Omron CX-Programmer project NewProject (CX-Programmer 9.75)

# PLC NewPLC1: CJ2M CPU31
I/O table (CPU CJ2M-CPU31): rack 0 slot 11 CJ2M-EIP21

## Global symbols (name address type ; comment)
0.00 BOOL  ; SW1
0.01 BOOL  ; CAPACITIVE 2
0.02 BOOL  ; CAPACITIVE 3
0.04 BOOL  ; INDUCTIVE SENSOR
0.13 BOOL  ; REEST PASS DENY
0.14 BOOL  ; RESET ACCESSS
0.15 BOOL  ; RESET ACCESS
10.00 BOOL  ; SW1
10.01 BOOL  ; SW2
10.02 BOOL  ; SW3
10.03 BOOL  ; SW4
10.04 BOOL  ; RESET
10.05 BOOL  ; START
10.06 BOOL  ; STOP
1.00 BOOL  ; MAS
1.01 BOOL  ; LED
1.02 BOOL  ; ACUATOR
1.03 BOOL  ; INDUCTIVE OUTPUT
1.04 BOOL  ; GREEN LIGHT
1.05 BOOL  ; RED LIGHT
1.07 BOOL  ; NOT MAS
1.08 BOOL  ; KA sw
1.15 BOOL  ; ACCESS DENIED
20.00 BOOL  ; K1
20.01 BOOL  ; K3
20.02 BOOL  ; K2
20.03 BOOL  ; K4
20.04 BOOL  ; ACCESS GRANTED
20.05 BOOL  ; KEEP 1
20.06 BOOL  ; KEEP SW2
30.00 BOOL  ; KS1
30.01 BOOL  ; KS2
30.02 BOOL  ; KS3
30.03 BOOL  ; KS4
40.00 BOOL  ; KA
40.01 BOOL  ; KB
40.02 BOOL  ; KC
40.03 BOOL  ; KD
40.04 BOOL  ; KEEP LIGHT1
C0000 BOOL  ; COUNTER PEPLE
C1 CHANNEL  ; compare

## Program NewProgram1 (cyclic task 0)
Local symbols
FSAFASF BOOL

### Section Section1

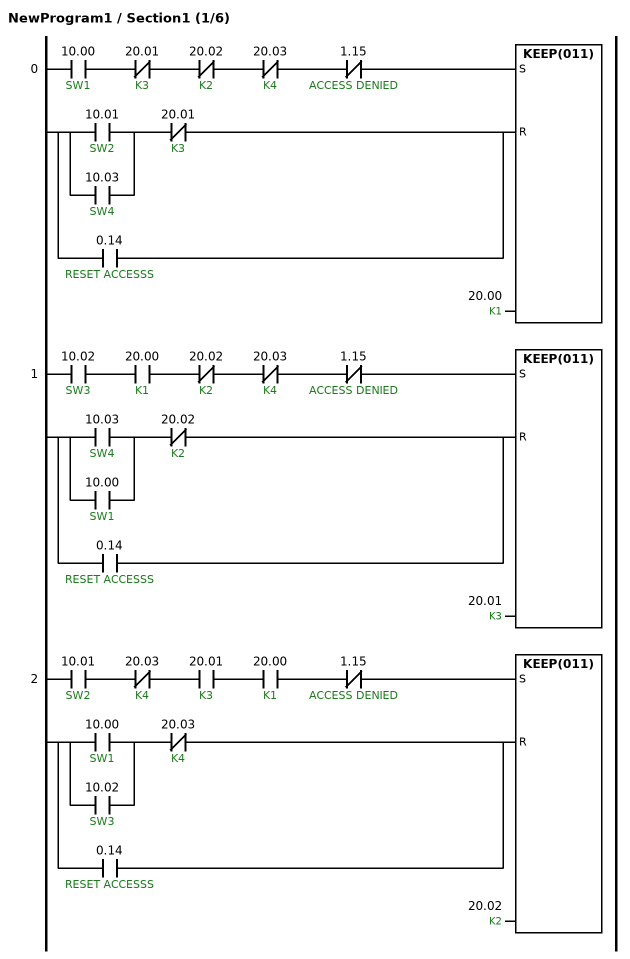
; rung 0
LD 10.00  ; SW1
ANDNOT 20.01  ; K3
ANDNOT 20.02  ; K2
ANDNOT 20.03  ; K4
ANDNOT 1.15  ; ACCESS DENIED
LD 10.01  ; SW2
OR 10.03  ; SW4
ANDNOT 20.01  ; K3
OR 0.14  ; RESET ACCESSS
KEEP(011) 20.00  ; K1
; rung 1
LD 10.02  ; SW3
AND 20.00  ; K1
ANDNOT 20.02  ; K2
ANDNOT 20.03  ; K4
ANDNOT 1.15  ; ACCESS DENIED
LD 10.03  ; SW4
OR 10.00  ; SW1
ANDNOT 20.02  ; K2
OR 0.14  ; RESET ACCESSS
KEEP(011) 20.01  ; K3
; rung 2
LD 10.01  ; SW2
ANDNOT 20.03  ; K4
AND 20.01  ; K3
AND 20.00  ; K1
ANDNOT 1.15  ; ACCESS DENIED
LD 10.00  ; SW1
OR 10.02  ; SW3
ANDNOT 20.03  ; K4
OR 0.14  ; RESET ACCESSS
KEEP(011) 20.02  ; K2

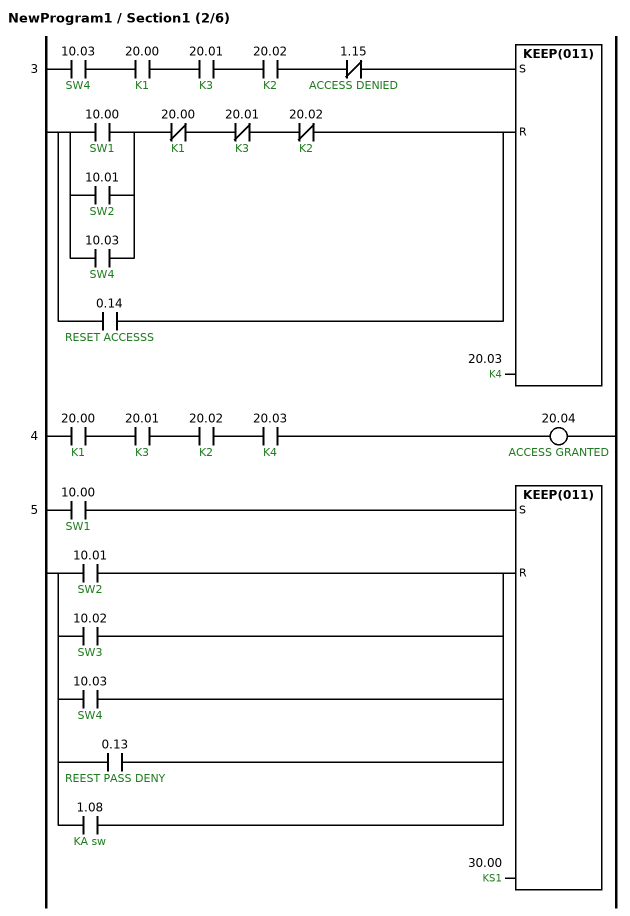
; rung 3
LD 10.03  ; SW4
AND 20.00  ; K1
AND 20.01  ; K3
AND 20.02  ; K2
ANDNOT 1.15  ; ACCESS DENIED
LD 10.00  ; SW1
OR 10.01  ; SW2
OR 10.03  ; SW4
ANDNOT 20.00  ; K1
ANDNOT 20.01  ; K3
ANDNOT 20.02  ; K2
OR 0.14  ; RESET ACCESSS
KEEP(011) 20.03  ; K4
; rung 4
LD 20.00  ; K1
AND 20.01  ; K3
AND 20.02  ; K2
AND 20.03  ; K4
OUT 20.04  ; ACCESS GRANTED
; rung 5
LD 10.00  ; SW1
LD 10.01  ; SW2
OR 10.02  ; SW3
OR 10.03  ; SW4
OR 0.13  ; REEST PASS DENY
OR 1.08  ; KA sw
KEEP(011) 30.00  ; KS1

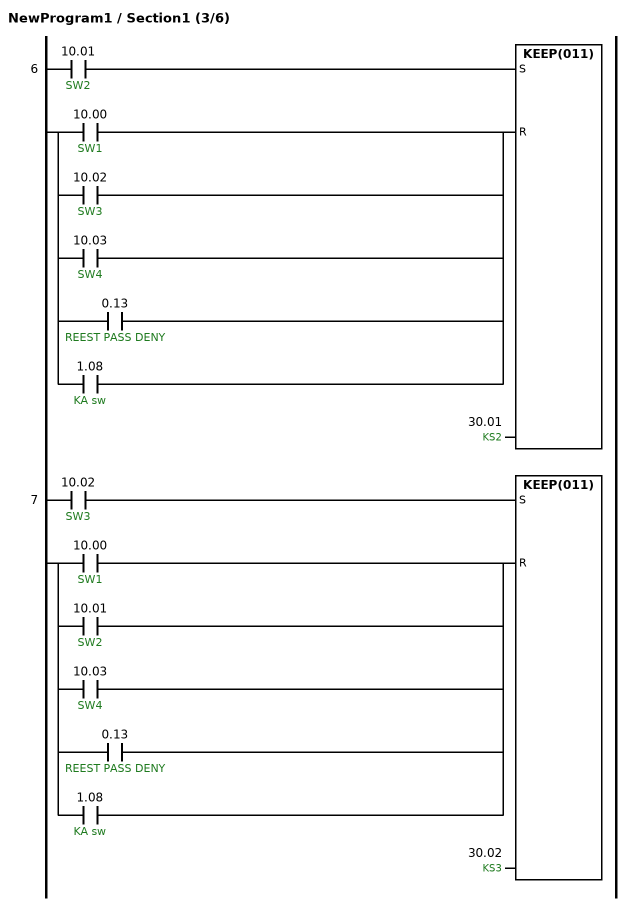
; rung 6
LD 10.01  ; SW2
LD 10.00  ; SW1
OR 10.02  ; SW3
OR 10.03  ; SW4
OR 0.13  ; REEST PASS DENY
OR 1.08  ; KA sw
KEEP(011) 30.01  ; KS2
; rung 7
LD 10.02  ; SW3
LD 10.00  ; SW1
OR 10.01  ; SW2
OR 10.03  ; SW4
OR 0.13  ; REEST PASS DENY
OR 1.08  ; KA sw
KEEP(011) 30.02  ; KS3

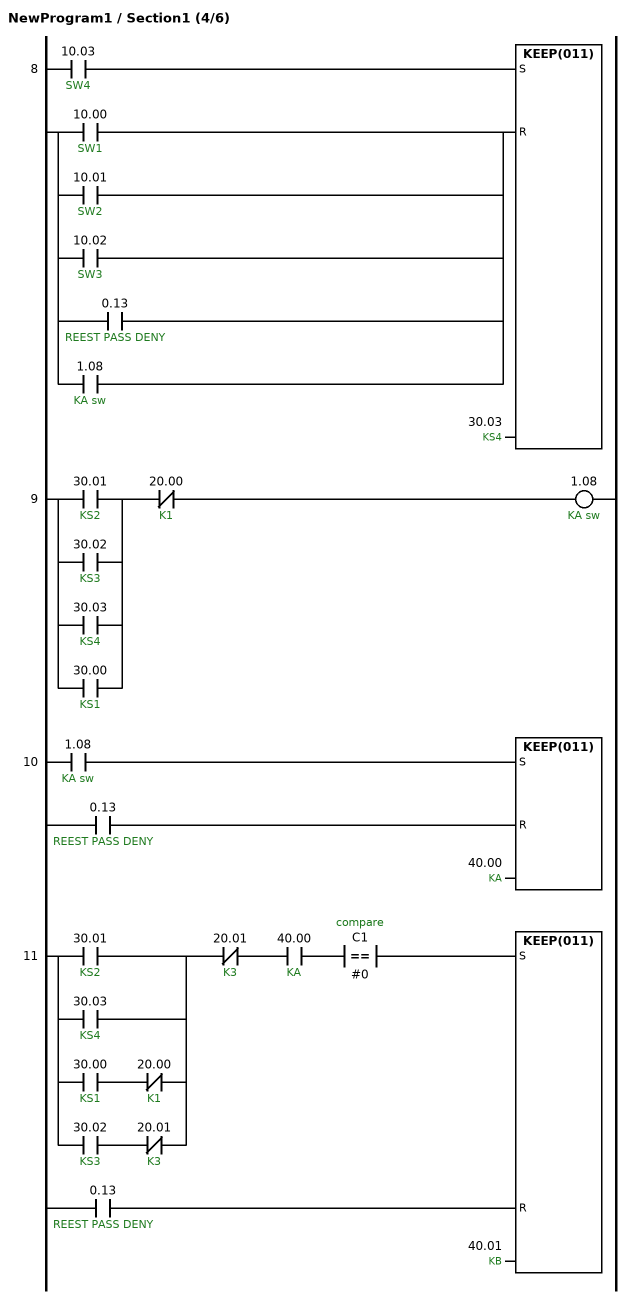
; rung 8
LD 10.03  ; SW4
LD 10.00  ; SW1
OR 10.01  ; SW2
OR 10.02  ; SW3
OR 0.13  ; REEST PASS DENY
OR 1.08  ; KA sw
KEEP(011) 30.03  ; KS4
; rung 9
LD 30.01  ; KS2
OR 30.02  ; KS3
OR 30.03  ; KS4
OR 30.00  ; KS1
ANDNOT 20.00  ; K1
OUT 1.08  ; KA sw
; rung 10
LD 1.08  ; KA sw
LD 0.13  ; REEST PASS DENY
KEEP(011) 40.00  ; KA
; rung 11
LD 30.01  ; KS2
OR 30.03  ; KS4
LD 30.00  ; KS1
ANDNOT 20.00  ; K1
ORLD
LD 30.02  ; KS3
ANDNOT 20.01  ; K3
ORLD
ANDNOT 20.01  ; K3
AND 40.00  ; KA
AND=(300) C1 #0  ; compare
LD 0.13  ; REEST PASS DENY
KEEP(011) 40.01  ; KB

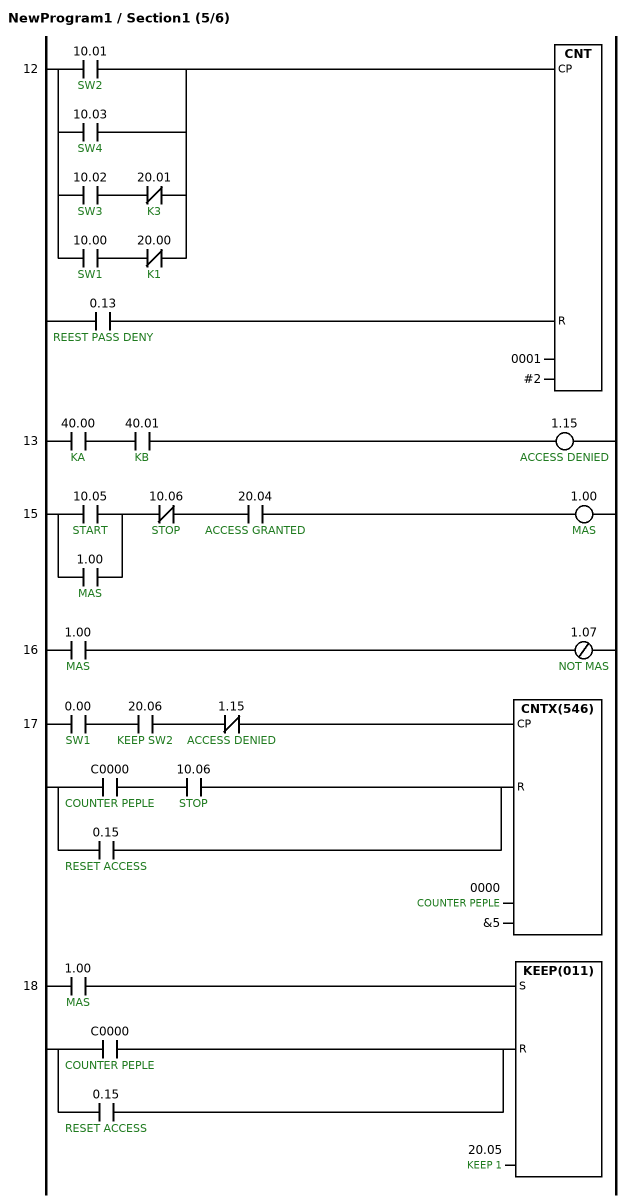
; rung 12
LD 10.01  ; SW2
OR 10.03  ; SW4
LD 10.02  ; SW3
ANDNOT 20.01  ; K3
ORLD
LD 10.00  ; SW1
ANDNOT 20.00  ; K1
ORLD
LD 0.13  ; REEST PASS DENY
CNT 0001 #2
; rung 13
LD 40.00  ; KA
AND 40.01  ; KB
OUT 1.15  ; ACCESS DENIED
; rung 15
LD 10.05  ; START
OR 1.00  ; MAS
ANDNOT 10.06  ; STOP
AND 20.04  ; ACCESS GRANTED
OUT 1.00  ; MAS
; rung 16
LD 1.00  ; MAS
OUTNOT 1.07  ; NOT MAS
; rung 17
LD 0.00  ; SW1
AND 20.06  ; KEEP SW2
ANDNOT 1.15  ; ACCESS DENIED
LD C0000  ; COUNTER PEPLE
AND 10.06  ; STOP
OR 0.15  ; RESET ACCESS
CNTX(546) 0000 &5  ; COUNTER PEPLE
; rung 18
LD 1.00  ; MAS
LD C0000  ; COUNTER PEPLE
OR 0.15  ; RESET ACCESS
KEEP(011) 20.05  ; KEEP 1

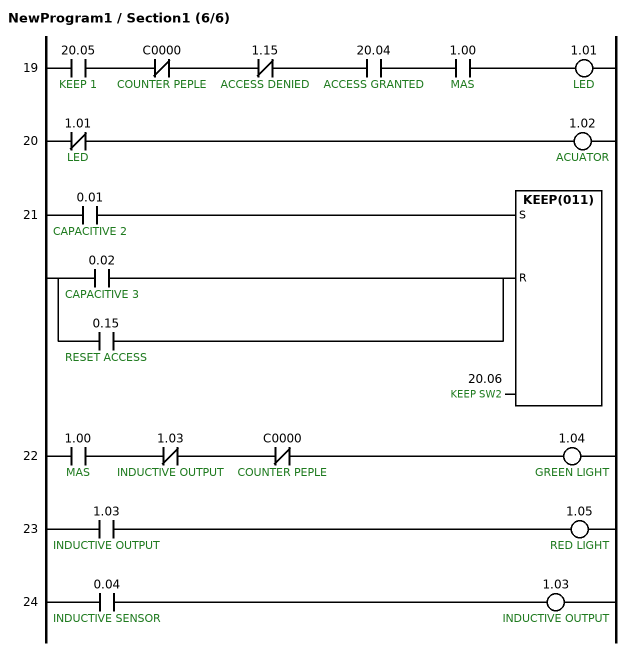
; rung 19
LD 20.05  ; KEEP 1
ANDNOT C0000  ; COUNTER PEPLE
ANDNOT 1.15  ; ACCESS DENIED
AND 20.04  ; ACCESS GRANTED
AND 1.00  ; MAS
OUT 1.01  ; LED
; rung 20
LDNOT 1.01  ; LED
OUT 1.02  ; ACUATOR
; rung 21
LD 0.01  ; CAPACITIVE 2
LD 0.02  ; CAPACITIVE 3
OR 0.15  ; RESET ACCESS
KEEP(011) 20.06  ; KEEP SW2
; rung 22
LD 1.00  ; MAS
ANDNOT 1.03  ; INDUCTIVE OUTPUT
ANDNOT C0000  ; COUNTER PEPLE
OUT 1.04  ; GREEN LIGHT
; rung 23
LD 1.03  ; INDUCTIVE OUTPUT
OUT 1.05  ; RED LIGHT
; rung 24
LD 0.04  ; INDUCTIVE SENSOR
OUT 1.03  ; INDUCTIVE OUTPUT

### Section END
; rung 0
END(001)